TYPE ST_Pointer_Data :
STRUCT
END_STRUCT
END_TYPE

(* stored: Version 1.1.0.1, ProductVersion 3.1.4026.17
   DUT ST_Pointer_Data: Id {82a05289-e64b-4e00-a876-a9f744e78869} *)
